// SIMATIC S7-200 project (STEP 7-Micro/WIN), CPU 224 REL 02.01

SYMBOL_TABLE 用户定义1
I0_0             I0.0     // 输入信号
I0_1             I0.1     // 设备运行信号
M0_0             M0.0     // 输入信号上升延微分
M0_1             M0.1     // 输入信号有效上升延微分
M14_1            M14.1    // 第1路输入信号保持状态
M14_2            M14.2    // 第2路输入信号保持状态
M14_3            M14.3    // 第3路输入信号保持状态
M16_1            M16.1    // 延迟输出保持状态
Q0_0             Q0.0     // 延迟输出信号
T_11             T11      // 延迟输出时间
T_12             T12      // 延迟输出时间
T_13             T13      // 延迟输出时间
T_91             T91      // 延迟输出保持时间
END_SYMBOL_TABLE

ORGANIZATION_BLOCK 主程序:OB1
TITLE=该程序可以实现输入延迟一定时间后输出，但延时输出时不再现输入动作时间，只输出一个动作信号；
// 该程序具有断电保持功能。
// 该程序为记忆3个输入信号的示例程序：最多可以同时记忆3个输入信号，其余的输入信号将会被忽略；也就是说，如果延迟输出时间为X秒，那么在任意一个X秒的时间段范围以内，最多只能有3个输入信号有效（被记忆），其余的输入信号将会被忽略；
// 如果希望记忆N个输入信号，将程序进行相应扩展即可；
// 对于每个输入信号而言，其延迟输出时间都是一样的，否则就没有任何意义了（从逻辑上来说，根本无法对某个指定的输入信号分配延迟输出时间）；
// 该示例程序的延迟输出时间为10秒，控制精度为0.1S；如果希望控制精度更高、延迟输出时间更长，请采用相应的定时器；如果无法找到合适的定时器，请采用和控制精度级别相同的定时器+多个计数器级联来实现。
BEGIN
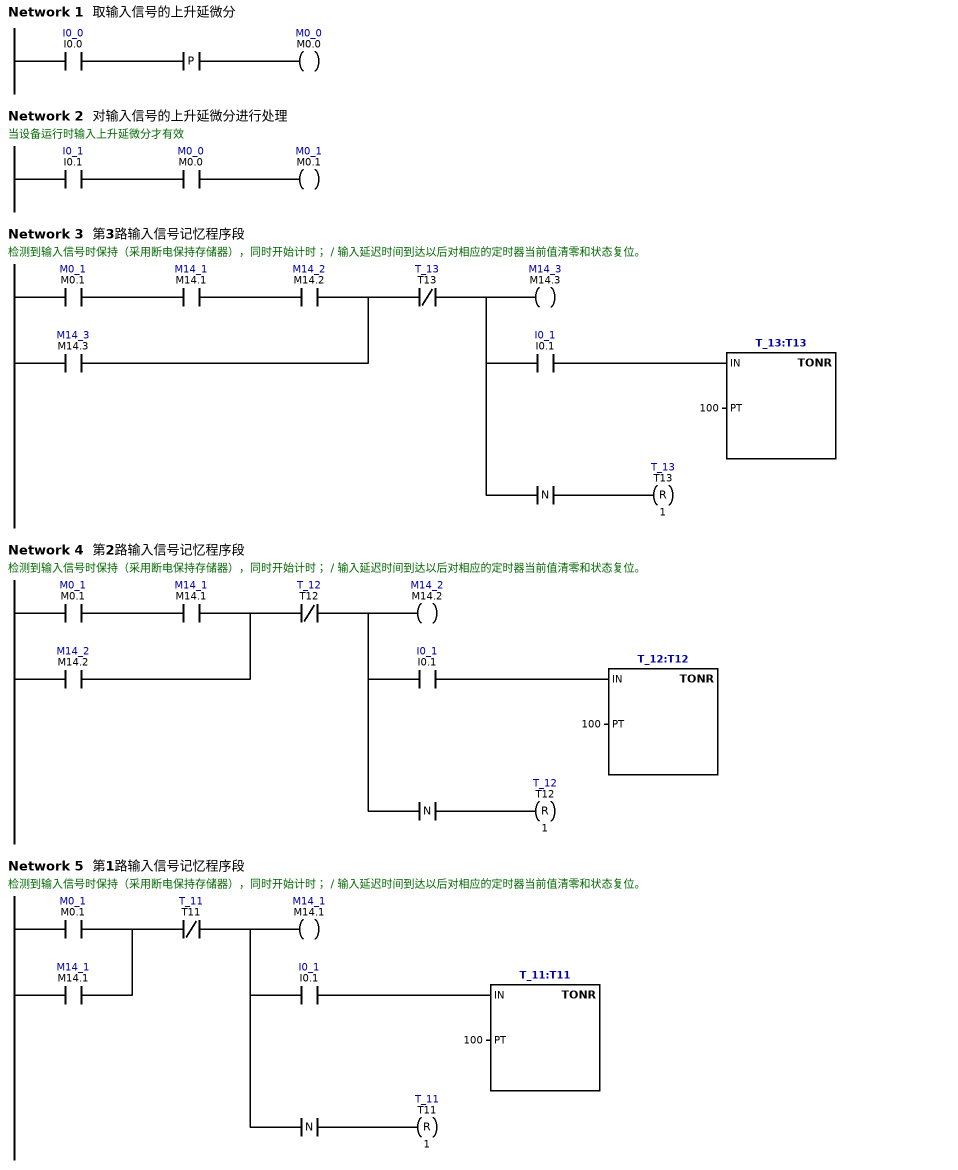
Network 1 // 取输入信号的上升延微分
LD     I0_0:I0.0
EU
=      M0_0:M0.0
Network 2 // 对输入信号的上升延微分进行处理
// 当设备运行时输入上升延微分才有效
LD     I0_1:I0.1
A      M0_0:M0.0
=      M0_1:M0.1
Network 3 // 第3路输入信号记忆程序段
// 检测到输入信号时保持（采用断电保持存储器），同时开始计时；
// 输入延迟时间到达以后对相应的定时器当前值清零和状态复位。
LD     M0_1:M0.1
A      M14_1:M14.1
A      M14_2:M14.2
O      M14_3:M14.3
AN     T_13:T13
LPS
=      M14_3:M14.3
A      I0_1:I0.1
TONR   T_13:T13, 100
LPP
ED
R      T_13:T13, 1
Network 4 // 第2路输入信号记忆程序段
// 检测到输入信号时保持（采用断电保持存储器），同时开始计时；
// 输入延迟时间到达以后对相应的定时器当前值清零和状态复位。
LD     M0_1:M0.1
A      M14_1:M14.1
O      M14_2:M14.2
AN     T_12:T12
LPS
=      M14_2:M14.2
A      I0_1:I0.1
TONR   T_12:T12, 100
LPP
ED
R      T_12:T12, 1
Network 5 // 第1路输入信号记忆程序段
// 检测到输入信号时保持（采用断电保持存储器），同时开始计时；
// 输入延迟时间到达以后对相应的定时器当前值清零和状态复位。
LD     M0_1:M0.1
O      M14_1:M14.1
AN     T_11:T11
LPS
=      M14_1:M14.1
A      I0_1:I0.1
TONR   T_11:T11, 100
LPP
ED
R      T_11:T11, 1
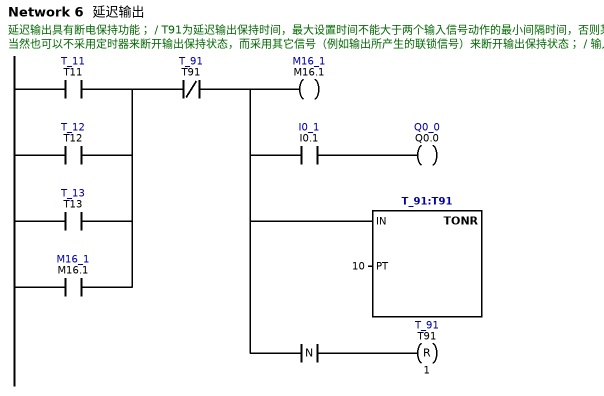
Network 6 // 延迟输出
// 延迟输出具有断电保持功能；
// T91为延迟输出保持时间，最大设置时间不能大于两个输入信号动作的最小间隔时间，否则某些输入信号将会被忽略而不会再现到输出；
// 当然也可以不采用定时器来断开输出保持状态，而采用其它信号（例如输出所产生的联锁信号）来断开输出保持状态；
// 输入断开以后对相应的定时器当前值清零和状态复位。
LD     T_11:T11
O      T_12:T12
O      T_13:T13
O      M16_1:M16.1
AN     T_91:T91
LPS
=      M16_1:M16.1
A      I0_1:I0.1
=      Q0_0:Q0.0
LRD
TONR   T_91:T91, 10
LPP
ED
R      T_91:T91, 1
END_ORGANIZATION_BLOCK
